(* CoDeSys 2.3 export: SIZE.EXP *)

(* Data type in INT *)
TYPE Size : UINT;
END_TYPE
